FUNCTION_BLOCK CHECKPOINT_DATA_GENERATOR (* Composite Function Block Type *)
  (* Standard: 61499-2 *)
  (* Version 0.0, 12/17/2022, Dmitrii, Flexbridge AB, template *)
  PACKAGE UAO.Hackathon;
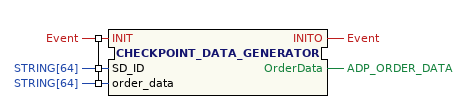
  EVENT_INPUT
    INIT WITH SD_ID, order_data;
  END_EVENT
  EVENT_OUTPUT
    INITO;
  END_EVENT
  VAR_INPUT
    SD_ID : STRING[64];
    order_data : STRING[64]; (* Indication Data from Plug *)
  END_VAR
  PLUGS
    OrderData : ADP_ORDER_DATA;
  END_PLUGS
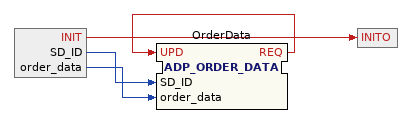
  EVENT_CONNECTIONS
    INIT TO INITO;
    OrderData.REQ TO OrderData.UPD;
  END_CONNECTIONS
  DATA_CONNECTIONS
    SD_ID TO OrderData.SD_ID;
    order_data TO OrderData.order_data;
  END_CONNECTIONS
END_FUNCTION_BLOCK
